Staubli VAL3: Form_Product.pgx

public program Form_Product(string x_sTitle, string& x_sLableList[], string& x_sList[], string x_sBottom)
  local num l_nNum
begin

//cls()
title(x_sTitle)
setTextMode(0)
for l_nNum=0 to size(x_sLableList)-1
  gotoxy(0,l_nNum+1)
  if l_nNum==2
    setTextMode(2)
  endIf
  put(left(x_sLableList[l_nNum]+"            ",18))
  setTextMode(0)
  gotoxy(22,l_nNum+1)

   put(left(x_sList[l_nNum]+"            ",18))
endFor

call Control_BottomS(x_sBottom)



end
